// TIA Portal V19 export
FUNCTION "HMI" : Void   // FC4, LAD
{ S7_Optimized_Access := 'TRUE' }
// stored: SetENOAutomatically false
BEGIN

REGION Network 1
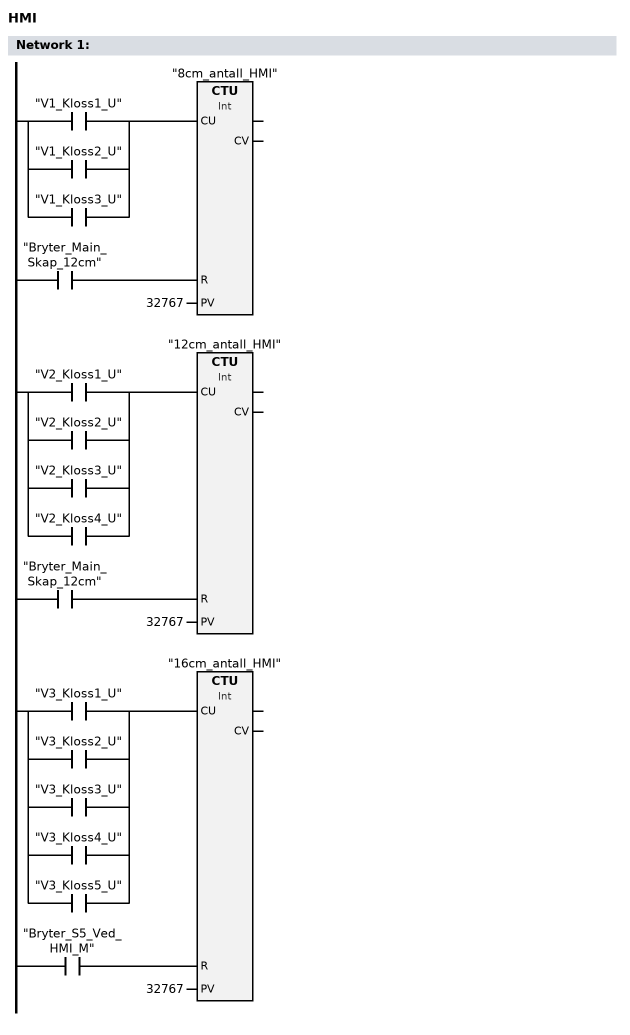
   RUNG wire#powerrail
      Contact( "V1_Kloss1_U" )
      wire#w1
      { S7_Templates := "value_type := Int" } "8cm_antall_HMI".CTU(r := wire#w2, pv := 32767, cv =>)
   END_RUNG
   RUNG wire#powerrail
      Contact( "V1_Kloss2_U" )
   END_RUNG wire#w1
   RUNG wire#powerrail
      Contact( "V1_Kloss3_U" )
   END_RUNG wire#w1
   RUNG wire#powerrail
      Contact( "Bryter_Main_Skap_12cm" )
   END_RUNG wire#w2
   RUNG wire#powerrail
      Contact( "V2_Kloss1_U" )
      wire#w3
      { S7_Templates := "value_type := Int" } "12cm_antall_HMI".CTU(r := wire#w4, pv := 32767, cv =>)
   END_RUNG
   RUNG wire#powerrail
      Contact( "V2_Kloss2_U" )
   END_RUNG wire#w3
   RUNG wire#powerrail
      Contact( "V2_Kloss3_U" )
   END_RUNG wire#w3
   RUNG wire#powerrail
      Contact( "V2_Kloss4_U" )
   END_RUNG wire#w3
   RUNG wire#powerrail
      Contact( "Bryter_Main_Skap_12cm" )
   END_RUNG wire#w4
   RUNG wire#powerrail
      Contact( "V3_Kloss1_U" )
      wire#w5
      { S7_Templates := "value_type := Int" } "16cm_antall_HMI".CTU(r := wire#w6, pv := 32767, cv =>)
   END_RUNG
   RUNG wire#powerrail
      Contact( "V3_Kloss2_U" )
   END_RUNG wire#w5
   RUNG wire#powerrail
      Contact( "V3_Kloss3_U" )
   END_RUNG wire#w5
   RUNG wire#powerrail
      Contact( "V3_Kloss4_U" )
   END_RUNG wire#w5
   RUNG wire#powerrail
      Contact( "V3_Kloss5_U" )
   END_RUNG wire#w5
   RUNG wire#powerrail
      Contact( "Bryter_S5_Ved_HMI_M" )
   END_RUNG wire#w6
   // the same network as SCL:
   "8cm_antall_HMI".CTU(CU := "V1_Kloss1_U" OR "V1_Kloss2_U" OR "V1_Kloss3_U",
                        R := "Bryter_Main_Skap_12cm",
                        PV := 32767);
   "12cm_antall_HMI".CTU(CU := "V2_Kloss1_U" OR "V2_Kloss2_U" OR "V2_Kloss3_U" OR "V2_Kloss4_U",
                         R := "Bryter_Main_Skap_12cm",
                         PV := 32767);
   "16cm_antall_HMI".CTU(CU := "V3_Kloss1_U" OR "V3_Kloss2_U" OR "V3_Kloss3_U" OR "V3_Kloss4_U" OR "V3_Kloss5_U",
                         R := "Bryter_S5_Ved_HMI_M",
                         PV := 32767);
END_REGION
END_FUNCTION
